(* IEC 61131-3 sources: test/src-senvion_wtt_ctl-plc/InterTaskCommunication, 3 files *)

(* ---- GetHandles.st ---- *)
PROGRAM GetHandles
VAR CONSTANT
	NbrOfHandleBlocks 	: INT := 2;
END_VAR
VAR
	i 				: INT;
	ErrMsgDone		: BOOL;
END_VAR
VAR_OUTPUT
	InitDone		: BOOL;
END_VAR

i := i + 1;

IF(i > NbrOfHandleBlocks)THEN
	i :=1;
END_IF

(* -------------------------------------------------------------------------------------------- *)
(* --- Get handles from WTT_IO - program max. 10 handles in each block *)
(* -------------------------------------------------------------------------------------------- *)

CASE i OF
	1:
		Handles.Example1 := WTTL_GetPresHd(LogicalNodeName := 'WTUR', DataObjectName := 'Example1' , CalcPer := 0);

	2:
		Handles.Example2 := WTTL_GetPresHd(LogicalNodeName := 'WTUR', DataObjectName := 'Example2' , CalcPer := 0);

END_CASE

(* -------------------------------------------------------------------------------------------- *)
(* --- Check handles *)
(* -------------------------------------------------------------------------------------------- *)
IF	(Handles.Example1 <> 0) AND
	(Handles.Example2 <> 0)
THEN
	InitDone := TRUE;
END_IF

IF NOT(InitDone) AND NOT(ErrMsgDone) AND (i = NbrOfHandleBlocks) THEN
	Util_LogErr('Error during initialization of the handles for WTT_CTL');
	ErrMsgDone := TRUE;
END_IF

END_PROGRAM

(* ---- TaskComMain.st ---- *)
PROGRAM TaskComMain
VAR
	IntMainToCtl			: MainToCtl;
	IntCtlToMain			: CtlToMain;
	ChkCnt					: DINT;
	MainToCtrlChkCntErr		: DINT;

	Parameter1 	: REAL;
	Parameter2 	: REAL;
	Parameter3 	: REAL;
	Parameter4 	: REAL;
	Parameter5 	: REAL;
	Parameter6 	: REAL;
	Wert1	   	: BOOL;
	Wert2		: INT;
	Wert3		: REAL;
	Wert4		: BOOL;
	Wert5		: REAL;

END_VAR

(* -------------------------------------------------------------------*)
(* -- Data from WTT_CTL to WTT_MAIN                                --*)
(* -------------------------------------------------------------------*)
ChkCnt := ChkCnt + 1;

IntCtlToMain.ChkCntStart := ChkCnt;
IntCtlToMain.Wert1 := TRUE;
IntCtlToMain.Wert2 := 22;
IntCtlToMain.Wert3 := 23;
IntCtlToMain.Wert4 := TRUE;
IntCtlToMain.Wert5 := 25;
IntCtlToMain.ChkCntEnd := ChkCnt;

Mem_AtomicCopy(Dst := ADR(CtlToMain), Src := ADR(IntCtlToMain), Len := SIZEOF(CtlToMain));

(* -------------------------------------------------------------------*)
(* -- Data from WTT_MAIN to WTT_CTL                                 --*)
(* -------------------------------------------------------------------*)

Mem_AtomicCopy(Dst := ADR(IntMainToCtl), Src := ADR(MainToCtl), Len := SIZEOF(MainToCtl));

IF(IntMainToCtl.ChkCntStart = IntMainToCtl.ChkCntEnd)THEN

	Parameter1 := IntMainToCtl.Parameter1;
	Parameter2 := IntMainToCtl.Parameter2;
	Parameter3 := IntMainToCtl.Parameter3;
	Parameter4 := IntMainToCtl.Parameter4;
	Parameter5 := IntMainToCtl.Parameter5;
	Parameter6 := IntMainToCtl.Parameter6;
	Wert1 := IntMainToCtl.Wert1;
	Wert2 := IntMainToCtl.Wert2;
	Wert3 := IntMainToCtl.Wert3;
	Wert4 := IntMainToCtl.Wert4;
	Wert5 := IntMainToCtl.Wert5;

ELSE
	MainToCtrlChkCntErr := MainToCtrlChkCntErr + 1;
END_IF

END_PROGRAM

(* ---- TaskComWtt.st ---- *)
PROGRAM TaskComWtt
VAR

END_VAR

MyExample := WTTL_GetMV( Hd := Handles.Example1);

END_PROGRAM
